(* PLC project  *)

CONFIGURATION EL2904
END_CONFIGURATION
